Staubli VAL3: _alter_stauts.pgx

program _alter_stauts()
begin
  while true
    gotoxy(0,12)
    put("* nAlter: "+toString("",nAlter)+"   ")
    gotoxy(12,12)
    put("* nAlterBegin: "+toString("",nAlterBegin)+"   ")
    delay(1)
  endWhile
end
